(* IEC 61131-3 sources: StCore/, 3 files *)

(* ---- StCore.typ ---- *)
(*******************************************************************************
 * File: StCore.typ
 * Author: Tyler Matijevich
 * Date: 2022-02-26
*******************************************************************************)

TYPE
	StCoreSystemInfoType : 	STRUCT  (*Extended system information*)
		Warnings : UDINT; (*(Par 1460) Active SuperTrak system warnings*)
		Faults : UDINT; (*(Par 1460) Active SuperTrak system faults*)
		SectionCount : USINT; (*(Par 1080) Section count*)
		Enabled : BOOL; (*(Derived) All sections are enabled*)
		Disabled : BOOL; (*(Derived) All sections are disabled*)
		MotorPower : BOOL; (*(Derived) All sections' motor voltage within range*)
		DisabledExternally : BOOL; (*(Derived) One or more section disabled from external condition*)
		SectionWarningPresent : BOOL; (*(Derived) One or more active SuperTrak section warning*)
		SectionFaultPresent : BOOL; (*(Derived) One or more active SuperTrak section fault*)
		PalletRecoveringCount : USINT; (*(Derived) Total number of pallets reporting recovering status*)
		PalletInitializingCount : USINT; (*(Derived) Total number of palelts reporting initializing (moving to load target) status*)
	END_STRUCT;
	StCoreSystemInternalType : 	STRUCT  (*Local internal system information*)
		State : USINT; (*Execution state*)
		PreviousErrorReset : BOOL; (*Previous ErrorReset value*)
	END_STRUCT;
	StCoreSectionInfoType : 	STRUCT  (*Extended section information*)
		Warnings : UDINT; (*(Par 1480) Active SuperTrak section warnings*)
		Faults : UDINT; (*(Par 1480) Active SuperTrak section faults*)
		PalletCount : USINT; (*(Par 1502) Number of pallets on the section*)
	END_STRUCT;
	StCoreSectionInternalType : 	STRUCT  (*Local internal section information*)
		State : USINT; (*Execution state*)
		PreviousErrorReset : BOOL; (*Previous ErrorReset value*)
	END_STRUCT;
	StCoreFunctionInternalType : 	STRUCT  (*Local internal function information*)
		State : USINT; (*Execution state*)
		Select : USINT; (*Select index (Section, Target, or Pallet)*)
		PreviousSelect : USINT; (*Previous select index value*)
		PreviousErrorReset : BOOL; (*Previous ErrorReset value*)
		PreviousCommand : UINT; (*Previous command inputs bitwise*)
		CommandSelect : USINT; (*Active command index*)
		pCommand : UDINT; (*Address of buffered core command*)
	END_STRUCT;
	StCoreTargetParameterType : 	STRUCT  (*Target interface parameters*)
		Release : StCoreReleaseParameterType; (*Release command parameters*)
		PalletID : USINT := 1; (*Pallet ID to assign*)
		Motion : StCoreMotionParameterType; (*Motion parameters for configuration command*)
		Mechanical : StCoreMechanicalParameterType; (*Mechanical parameters for configuration command*)
		Control : StCoreControlParameterType; (*Control parameters for configuration command*)
	END_STRUCT;
	StCoreReleaseParameterType : 	STRUCT  (*Release command parameter structure*)
		Direction : UINT := stDIRECTION_RIGHT; (*Direction of motion (stDIRECTION_RIGHT or stDIRECTION_LEFT)*)
		DestinationTarget : USINT := 1; (*Destination target*)
		Offset : LREAL; (*(mm) [-500, 500] Target offset or incremental offset*)
	END_STRUCT;
	StCoreMotionParameterType : 	STRUCT  (*Motion parameter structure*)
		Velocity : REAL; (*(mm/s) [5, 4000] Set velocity*)
		Acceleration : REAL; (*(mm/s/s) [500, 60000] Set acceleration and deceleration*)
	END_STRUCT;
	StCoreMechanicalParameterType : 	STRUCT  (*Mechanical parameter structure*)
		ShelfWidth : LREAL; (*(mm) [152, 600] Physical pallet shelf length*)
		CenterOffset : LREAL; (*(mm) Physical pallet shelf center offset*)
	END_STRUCT;
	StCoreControlParameterType : 	STRUCT  (*Control parameter structure*)
		ControlGainSet : USINT; (*[0, 15] Select control gain set*)
		MovingFilter : REAL := 0.5; (*[0, 1) Moving control filter weight*)
		StationaryFilter : REAL := 0.5; (*[0, 1) Stationary control filter weight*)
	END_STRUCT;
	StCoreTargetInfoType : 	STRUCT  (*Extended target information*)
		Section : USINT; (*(Par 1650) Target section number*)
		Position : LREAL; (*mm (Derived) Target section position*)
		PositionUm : DINT; (*um (Par 1651) Target integer section position*)
		PalletCount : USINT; (*(Derived) The number of pallets destined to this target*)
	END_STRUCT;
	StCoreTargetStatusType : 	STRUCT  (*Target status information*)
		PalletPresent : BOOL; (*(IF) A pallet has arrived, entered the in-position window, and is not yet released*)
		PalletInPosition : BOOL; (*(IF) A pallet is currently within the in-position window*)
		PalletPreArrival : BOOL; (*(IF) A pallet is expected to arrive at the stop within the configured time*)
		PalletOverTarget : BOOL; (*(IF) A pallet's shelf is over the target (requires configuration to report status)*)
		PalletPositionUncertain : BOOL; (*(IF) A pallet has arrived but is not reporting in-position*)
		PalletID : USINT; (*(IF) ID of the pallet present at the target*)
		Info : StCoreTargetInfoType; (*Extended target status information*)
	END_STRUCT;
END_TYPE

(* ---- StCore.fun ---- *)
(*******************************************************************************
 * File: StCore.fun
 * Author: Tyler Matijevich
 * Date: 2022-02-15
*******************************************************************************)
(*SuperTrak control program*)

FUNCTION StCoreInit : DINT (*Initialize SuperTrak, verify layout, read targets, and size control interface*)
	VAR_INPUT
		StoragePath : STRING[127]; (*Filesystem location for SuperTrak configuration data*)
		SimIPAddress : STRING[15]; (*CPU configuration's simulation IP address*)
		EthernetInterfaceList : STRING[63]; (*Comma-separated list of ethernet interfaces ('IF3,IF4')*)
		PalletCount : USINT; (*Maximum number of pallets on system*)
		NetworkIOCount : USINT; (*Maximum number of network I/O channels on system*)
	END_VAR
END_FUNCTION

FUNCTION StCoreCyclic : DINT (*Process SuperTrak control interface*)
END_FUNCTION

FUNCTION StCoreExit : DINT (*Free internal memory*)
END_FUNCTION
(*******************************************************************************
SuperTrak control interface
*******************************************************************************)
(*System and sections*)

FUNCTION_BLOCK StCoreSystem (*SuperTrak system interface function*)
	VAR_INPUT
		Enable : BOOL; (*Enable function execution*)
		ErrorReset : BOOL; (*Reset function error*)
		Debug : BOOL; (*Enable debug messages of command interface*)
		EnableAllSections : BOOL; (*(IF) Enable all sections*)
		AcknowledgeFaults : BOOL; (*(IF) Clear SuperTrak system faults or warnings*)
	END_VAR
	VAR_OUTPUT
		Valid : BOOL; (*Successful interface function execution*)
		Error : BOOL; (*An error has occurred with the function*)
		StatusID : DINT; (*Function error identifier. See logger for more details*)
		PalletsStopped : BOOL; (*(IF) All pallets are currently not moving*)
		WarningPresent : BOOL; (*(IF) A system warning message has been recorded*)
		FaultPresent : BOOL; (*(IF) A system fault message has been recorded*)
		PalletCount : USINT; (*(IF) Total number of pallets on the system*)
		Info : StCoreSystemInfoType; (*Extended system information*)
	END_VAR
	VAR
		Internal : StCoreFunctionInternalType; (*Local internal data*)
	END_VAR
END_FUNCTION_BLOCK

FUNCTION_BLOCK StCoreSection (*SuperTrak section interface function*)
	VAR_INPUT
		Enable : BOOL; (*Enable function execution*)
		Section : USINT; (*Select section*)
		ErrorReset : BOOL; (*Reset function error*)
		EnableSection : BOOL; (*(IF) Enable section control*)
		AcknowledgeFaults : BOOL; (*(IF) Clear SuperTrak section faults or warnings*)
	END_VAR
	VAR_OUTPUT
		Valid : BOOL; (*Successful interface function execution*)
		Error : BOOL; (*An error has occurred with the function*)
		StatusID : DINT; (*Function error identifier. See logger for more details*)
		Enabled : BOOL; (*(IF) Section control is enabled*)
		UnrecognizedPallets : BOOL; (*(IF) Section has one or more pallets with undetermined position. The section will automatically jog these pallets to locate them*)
		MotorPowerOn : BOOL; (*(IF) Motor supply voltage is within range*)
		PalletsRecovering : BOOL; (*(IF) Pallets must return to their last controlled position*)
		LocatingPallets : BOOL; (*(IF) Section is automatically jogging pallets to determine their location*)
		DisabledExternally : BOOL; (*(IF) Section is disabled due to an external condition*)
		WarningPresent : BOOL; (*(IF) A section warning message has been recorded*)
		FaultPresent : BOOL; (*(IF) A section fault message has been recorded*)
		DisabledPallet : BOOL; (*(IF) The section has one or more open-loop pallets present*)
		PalletsInitializing : BOOL; (*(IF) Pallets are making their initial move to the Load Target*)
		Info : StCoreSectionInfoType; (*Extended section information*)
	END_VAR
	VAR
		Internal : StCoreFunctionInternalType; (*Local internal data*)
	END_VAR
END_FUNCTION_BLOCK
(*Simple target release*)

FUNCTION StCoreSimpleRelease : DINT (*Release with local move configuration*)
	VAR_INPUT
		Target : USINT; (*Target (with pallet present)*)
		LocalMove : USINT; (*Local move configuration 1, 2, or 3*)
	END_VAR
END_FUNCTION
(*Release commands*)

FUNCTION StCoreReleasePallet : DINT (*Release pallet to target*)
	VAR_INPUT
		Target : USINT; (*Target (with pallet present)*)
		Pallet : USINT; (*Pallet ID*)
		Direction : UINT; (*Direction of motion (stDIRECTION_RIGHT or stDIRECTION_LEFT)*)
		DestinationTarget : USINT; (*Destination target*)
	END_VAR
END_FUNCTION

FUNCTION StCoreReleaseTargetOffset : DINT (*Release pallet to target + offset*)
	VAR_INPUT
		Target : USINT; (*Target (with pallet present)*)
		Pallet : USINT; (*Pallet ID*)
		Direction : UINT; (*Direction of motion (stDIRECTION_RIGHT or stDIRECTION_LEFT)*)
		DestinationTarget : USINT; (*Destination target*)
		TargetOffset : LREAL; (*[-500.0, 500.0] mm Absolute offset from destination target*)
	END_VAR
END_FUNCTION

FUNCTION StCoreReleaseIncrementalOffset : DINT (*Increment pallet offset*)
	VAR_INPUT
		Target : USINT; (*Target with pallet present*)
		Pallet : USINT; (*Pallet ID*)
		IncrementalOffset : LREAL; (*[-500.0, 500.0] mm Relative offset from current destination*)
	END_VAR
END_FUNCTION

FUNCTION StCoreContinueMove : DINT (*Resume pallet movement when at mandatory stop*)
	VAR_INPUT
		Target : USINT; (*Target (with pallet present)*)
		Pallet : USINT; (*Pallet ID*)
	END_VAR
END_FUNCTION
(*Configuration commands*)

FUNCTION StCoreSetPalletID : DINT (*Set ID of pallet at target*)
	VAR_INPUT
		Target : USINT; (*Target (with pallet present)*)
		PalletID : USINT; (*Pallet ID to assign*)
	END_VAR
END_FUNCTION

FUNCTION StCoreSetMotionParameters : DINT (*Set pallet velocity and/or acceleration*)
	VAR_INPUT
		Target : USINT; (*Target (with pallet present)*)
		Pallet : USINT; (*Pallet ID*)
		Velocity : LREAL; (*mm/s Set velocity (0.0 for unchanged)*)
		Acceleration : LREAL; (*mm/s^2 Set acceleration (0.0 for unchanged)*)
	END_VAR
END_FUNCTION

FUNCTION StCoreSetMechanicalParameters : DINT (*Set pallet shelf width and offset*)
	VAR_INPUT
		Target : USINT; (*Target (with pallet present)*)
		Pallet : USINT; (*Pallet ID*)
		ShelfWidth : LREAL; (*mm*)
		CenterOffset : LREAL;
	END_VAR
END_FUNCTION

FUNCTION StCoreSetControlParameters : DINT (*Set pallet control parameters*)
	VAR_INPUT
		Target : USINT; (*Target (with pallet present)*)
		Pallet : USINT; (*Pallet ID*)
		ControlGainSet : USINT; (*[0, 15] Control gain set defined in TrakMaster*)
		MovingFilter : LREAL; (*[0.0, 1.0) Moving control weight filter*)
		StationaryFilter : LREAL; (*[0.0, 1.0) Stationary control weight filter*)
	END_VAR
END_FUNCTION
(*Targets and pallets*)

FUNCTION StCoreTargetStatus : DINT (*Get target status*)
	VAR_INPUT
		Target : USINT; (*Target number*)
	END_VAR
	VAR_IN_OUT
		Status : StCoreTargetStatusType; (*Target status reference*)
	END_VAR
END_FUNCTION

FUNCTION_BLOCK StCoreTarget (*Target core interface*)
	VAR_INPUT
		Enable : BOOL; (*Enable function execution*)
		Target : USINT; (*Select target*)
		ErrorReset : BOOL; (*Reset function error*)
		Parameters : StCoreTargetParameterType; (*Command parameters*)
		ReleasePallet : BOOL; (*Release pallet to a target*)
		ReleaseTargetOffset : BOOL; (*Release pallet to a target plus offset*)
		ReleaseIncrementalOffset : BOOL; (*Increment a pallet's current offset*)
		ContinueMove : BOOL; (*Resume a pallet's previously requested move when stopped*)
		SetPalletID : BOOL; (*Set the pallet's ID*)
		SetMotionParameters : BOOL; (*Set the pallet's velocity and acceleration*)
		SetMechanicalParameters : BOOL; (*Set the pallet's shelf width and center offset*)
		SetControlParameters : BOOL; (*Set the pallet's control gain set and filter weights*)
	END_VAR
	VAR_OUTPUT
		Valid : BOOL; (*Successful function execution*)
		Error : BOOL; (*An error has occurred with the function*)
		StatusID : DINT; (*Function error identifier*)
		PalletPresent : BOOL; (*(IF) A pallet has arrived, entered the in-position window, and is not yet released*)
		PalletInPosition : BOOL; (*(IF) A pallet is currently within the in-position window*)
		PalletPreArrival : BOOL; (*(IF) A pallet is expected to arrive at the stop within the configured time*)
		PalletOverTarget : BOOL; (*(IF) A pallet's shelf is over the target (requires configuration to report status)*)
		PalletPositionUncertain : BOOL; (*(IF) A pallet has arrived but is not reporting in-position*)
		PalletID : USINT; (*(IF) ID of the pallet present at the target*)
		Info : StCoreTargetInfoType; (*Extended target information*)
		Busy : BOOL; (*A command request is executing*)
		Acknowledged : BOOL; (*A command request has successfully acknowledged*)
	END_VAR
	VAR
		Internal : StCoreFunctionInternalType; (*Local internal data*)
	END_VAR
END_FUNCTION_BLOCK

FUNCTION StCorePalletStatus : DINT (*Get pallet status*)
	VAR_INPUT
		Pallet : USINT; (*Pallet ID*)
	END_VAR
	VAR_IN_OUT
		Status : StCorePalletStatusType; (*Pallet status reference*)
	END_VAR
END_FUNCTION

FUNCTION_BLOCK StCorePallet (*Pallet core interface*)
	VAR_INPUT
		Enable : BOOL; (*Enable function execution*)
		Pallet : USINT; (*Select pallet ID*)
		ErrorReset : BOOL; (*Reset function error*)
		Parameters : StCorePalletParameterType; (*Command parameters*)
		ReleasePallet : BOOL; (*Release pallet to a target*)
		ReleaseTargetOffset : BOOL; (*Release pallet to a target plus offset*)
		ReleaseIncrementalOffset : BOOL; (*Increment a pallet's current offset*)
		ContinueMove : BOOL; (*Resume a pallet's previously requested move when stopped*)
		SetMotionParameters : BOOL; (*Set the pallet's velocity and acceleration*)
		SetMechanicalParameters : BOOL; (*Set the pallet's shelf width and center offset*)
		SetControlParameters : BOOL; (*Set the pallet's control gain set and filter weights*)
	END_VAR
	VAR_OUTPUT
		Valid : BOOL; (*Successful function execution*)
		Error : BOOL; (*An error has occurred with the function*)
		StatusID : DINT; (*Function error identifier*)
		Present : BOOL; (*(Par 1328) Pallet is present on the system*)
		Recovering : BOOL; (*(Par 1328) Pallet requires recovery when enabled or is recovering*)
		AtTarget : BOOL; (*(Par 1328) Pallet has arrived at target and is in position*)
		InPosition : BOOL; (*(Par 1328) Pallet is in position at target*)
		ServoEnabled : BOOL; (*(Par 1328) Pallet is currently controlled by the system*)
		Initializing : BOOL; (*(Par 1328) Pallet is moving to Load Target*)
		Lost : BOOL; (*(Par 1328) Pallet has lost position feedback*)
		Section : USINT; (*(Par 1307) Actual pallet section number*)
		Position : LREAL; (*mm (Par 1310) Actual pallet position*)
		Info : StCorePalletInfoType; (*Extended pallet information*)
		Busy : BOOL; (*A command request is executing*)
		Acknowledged : BOOL; (*A command request has successfully acknowledged*)
	END_VAR
	VAR
		Internal : StCoreFunctionInternalType; (*Local internal data*)
	END_VAR
END_FUNCTION_BLOCK
(*Network IO*)

FUNCTION StCoreGetNetworkIO : DINT (*Get network IO (output)*)
	VAR_INPUT
		Offset : USINT; (*Network output offset*)
		pValue : REFERENCE TO BOOL; (*Reference output value*)
	END_VAR
END_FUNCTION

FUNCTION StCoreSetNetworkIO : DINT (*Set network IO (input)*)
	VAR_INPUT
		Offset : USINT; (*Network input offset*)
		Value : BOOL; (*Network input value*)
	END_VAR
END_FUNCTION

(* ---- StCore.var ---- *)
(*******************************************************************************
 * File: StCore.var
 * Author: Tyler Matijevich
 * Date: 2022-03-02
*******************************************************************************)
(*Initialization*)
VAR CONSTANT
	stCORE_ERROR_LOGBOOK : DINT := -536805912; (*An error occurred during initialization when creating the logbook*)
	stCORE_ERROR_INITIALIZATION : DINT := -536804376; (*StCoreInit has not been called*)
	stCORE_ERROR_LAYOUT : DINT := -536804276; (*Invalid SuperTrak layout due to the section count, section addresses, or network order*)
END_VAR
(*Cyclic*)
VAR CONSTANT
	stCORE_ERROR_CYCLE : DINT := -536803376; (*StCoreCyclic is not called from task class #1 or does not match cycle time of 800 us*)
	stCORE_ERROR_PROTOCAL : DINT := -536803276; (*SuperTrak control interface configuration modified from initialization*)
	stCORE_ERROR_PALLET : DINT := -536803176; (*An unallocated pallet has been discovered on the SuperTrak*)
END_VAR
(*Common*)
VAR CONSTANT
	stCORE_ERROR_PARAMETER : DINT := -536802376; (*SuperTrak service channel error*)
	stCORE_ERROR_ALLOCATION : DINT := -536802276; (*Unable to allocate or reference cyclic StCore data*)
END_VAR
(*Function*)
VAR CONSTANT
	stCORE_ERROR_CONTEXT : DINT := -536801376; (*StCore command context (target or pallet) does not exist on the system*)
	stCORE_ERROR_BUFFER : DINT := -536801276; (*StCore command request is rejected due to full buffer*)
	stCORE_WARNING_BUFFER : DINT := -1610543099; (*Future StCore command requests will be rejected until buffer empties*)
	stCORE_WARNING_CHANNEL : DINT := -1610543098; (*Pallet command buffers are paused because all channels are in use*)
	stCORE_ERROR_TIMEOUT : DINT := -536800976; (*StCore command response from SuperTrak has timed out*)
	stCORE_ERROR_COMMAND : DINT := -536800876; (*SuperTrak responded with error to StCore command request*)
END_VAR
(*Interface*)
VAR CONSTANT
	stCORE_ERROR_INSTANCE : DINT := -536800376; (*Multiple instances of the function block are used in the same context*)
	stCORE_ERROR_INDEX : DINT := -536800276; (*The user index selection (section, target, or pallet) does not exist on the system*)
	stCORE_WARNING_INDEX : DINT := -1610542099; (*The user index selection has been modified while the function block is enabled*)
	stCORE_ERROR_ACKNOWLEDGE : DINT := -536800176; (*StCore function block is unable to acknowledge the command request due to buffer overwrite*)
END_VAR
